FUNCTION_BLOCK PUBLIC Boolean IMPLEMENTS I_StepCondition
VAR_INPUT
END_VAR
VAR_OUTPUT
END_VAR
VAR
	bValue : BOOL;
END_VAR

PROPERTY getValue : BOOL
GET
getValue := bValue;
END_GET
END_PROPERTY


PROPERTY setValue : BOOL
SET
bValue := setValue;
END_SET
END_PROPERTY

END_FUNCTION_BLOCK

(* stored: Version 1.1.0.1, ProductVersion 3.1.4024.0
   POU Boolean: Id {5a25ad0f-0be9-40c2-a688-0b7e5ac06027}, SpecialFunc None
   Property getValue: Id {2ef472d3-2576-4eb6-86b5-a760f7cf25e3}
   Get Get: Id {b387bbd5-5b88-464d-8939-5b2f201fd48a}
   Property setValue: Id {6d88ed92-8dc0-4fa2-a3c1-f0af7a358ad9}
   Set Set: Id {4bcac0eb-fbde-4ecf-b327-e522662e0592} *)
